TYPE (* A Structure with 8 Bits *)
  (* Version 1.0, 2024-02-21, franz *)
  st08b : STRUCT
    b00 : BOOL; (* BIT 00 *)
    b01 : BOOL; (* BIT 01 *)
    b02 : BOOL; (* BIT 02 *)
    b03 : BOOL; (* BIT 03 *)
    b04 : BOOL; (* BIT 04 *)
    b05 : BOOL; (* BIT 05 *)
    b06 : BOOL; (* BIT 06 *)
    b07 : BOOL; (* BIT 07 *)
  END_STRUCT;
END_TYPE
